// TIA Portal project "VFD_CommFault" (V17)

(* hardware
DEVICE "PLC_1"  S7-1200 Station
   slot 0: "Rack_0"  S7-1200 Rack  Rack  V1.0
   slot 1: "PLC_1"  CPU 1214C AC/DC/Rly  6ES7 214-1BG40-0XB0  V4.5
*)

// ===== PLC "PLC_1"  CPU 1214C AC/DC/Rly =====

DATA_BLOCK "内部数据"   // DB1
{ S7_Optimized_Access := 'TRUE' }
VERSION : 0.1
   VAR
      变频器读取失败1 : Bool;   // 变频器读取失败标志
      变频器读取成功1 : Bool;   // 变频器读取成功标志
      变频器通讯故障脉冲1 : Bool;   // 变频器通讯故障上升沿脉冲1
      变频器通讯故障脉冲2 : Bool;   // 变频器通讯故障上升沿脉冲2
      变频器通讯故障标志 : Bool;   // 变频器通讯故障标志位
      变频器通讯延时定时器 : IEC_TIMER;   // 变频器通讯延时定时器3分钟
   END_VAR
BEGIN
END_DATA_BLOCK

DATA_BLOCK "曲线数据"   // DB2
{ S7_Optimized_Access := 'TRUE' }
VERSION : 0.1
   VAR
      变频器通讯故障 : Bool;   // 变频器通讯故障报警
   END_VAR
BEGIN
END_DATA_BLOCK

FUNCTION "FC_VFD_CommFault" : Void   // FC1, LAD
{ S7_Optimized_Access := 'TRUE' }
   VAR_TEMP   // added for the SCL form of the ladder/FBD networks
      _w1 : Bool;
      _w2 : Bool;
   END_VAR
BEGIN

REGION Network 1: 变频器通讯故障检测
   // 检测变频器通讯失败/成功的上升沿，置位/复位故障标志；若故障标志保持接通3分钟以上则输出通讯故障报警。
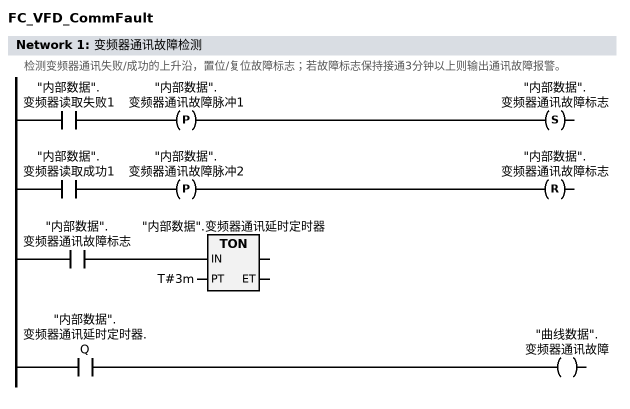
   #_w1 := "内部数据".变频器读取失败1 AND NOT "内部数据".变频器通讯故障脉冲1;   // rising edge
   "内部数据".变频器通讯故障脉冲1 := "内部数据".变频器读取失败1;
   IF #_w1 THEN "内部数据".变频器通讯故障标志 := TRUE; END_IF;
   #_w2 := "内部数据".变频器读取成功1 AND NOT "内部数据".变频器通讯故障脉冲2;   // rising edge
   "内部数据".变频器通讯故障脉冲2 := "内部数据".变频器读取成功1;
   IF #_w2 THEN "内部数据".变频器通讯故障标志 := FALSE; END_IF;
   "内部数据".变频器通讯延时定时器.TON(IN := "内部数据".变频器通讯故障标志, PT := T#3m);
   "曲线数据".变频器通讯故障 := "内部数据".变频器通讯延时定时器.Q;
END_REGION
END_FUNCTION

ORGANIZATION_BLOCK "Main"   // OB1, LAD, ProgramCycle
TITLE = "Main Program Sweep (Cycle)"
{ S7_Optimized_Access := 'TRUE' }
VERSION : 0.1
   VAR_INPUT
      Initial_Call : Bool;   // Initial call of this OB
      Remanence : Bool;   // =True, if remanent data are available
   END_VAR
BEGIN
END_ORGANIZATION_BLOCK